FUNCTION_BLOCK FB_Simu_AxisLIN_V1_1 EXTENDS FB_Simu_axis
VAR_INPUT

END_VAR
VAR_OUTPUT
END_VAR
VAR
END_VAR

rOUT_PixActual := MAP_REAL_TO_INT(rValue    := rIN_PosActual,
                                  rFromHigh := rIN_PosMax,
                                  rFromLow  := rIN_PosMin,
                                  rToHigh   := rIN_PixMax,
                                  rToLow    := rIN_PixMin);
(*
IF xIN_Enable THEN
    OUT_axis_ref := ADR(IN_axis_ref_simu);
ELSE
    OUT_axis_ref := ADR(IN_axis_ref);
END_IF
*)

END_FUNCTION_BLOCK

(* stored: Version 1.1.0.1, ProductVersion 3.1.4024.6
   POU FB_Simu_AxisLIN_V1_1: Id {6f3f35c2-88df-45cf-9274-41d0c42c68b0}, SpecialFunc None *)
